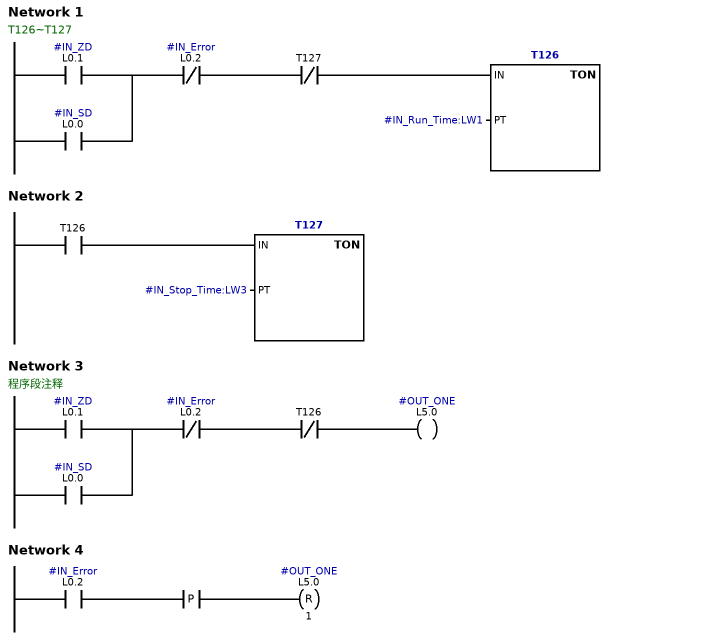
[picture p216: SBR112 networks 1-4]
Network 1
// T126~T127
LD     #IN_ZD:L0.1
O      #IN_SD:L0.0
AN     #IN_Error:L0.2
AN     T127
TON    T126, #IN_Run_Time:LW1
Network 2
LD     T126
TON    T127, #IN_Stop_Time:LW3
Network 3
// 程序段注释
LD     #IN_ZD:L0.1
O      #IN_SD:L0.0
AN     #IN_Error:L0.2
AN     T126
=      #OUT_ONE:L5.0
Network 4
LD     #IN_Error:L0.2
EU
R      #OUT_ONE:L5.0, 1
END_SUBROUTINE_BLOCK

SUBROUTINE_BLOCK Valve1_XH14:SBR113
TITLE=
VAR_INPUT
IN_SD:BOOL;	// L0.0 
IN_ZD:BOOL;	// L0.1 
IN_Error:BOOL;	// L0.2 
IN_Run_Time:INT;	// LW1 
IN_Stop_Time:INT;	// LW3 
END_VAR
VAR_OUTPUT
OUT_ONE:BOOL;	// L5.0 
END_VAR
VAR
TP1:BOOL;	// L5.1 
TP2:BOOL;	// L5.2 
END_VAR
BEGIN
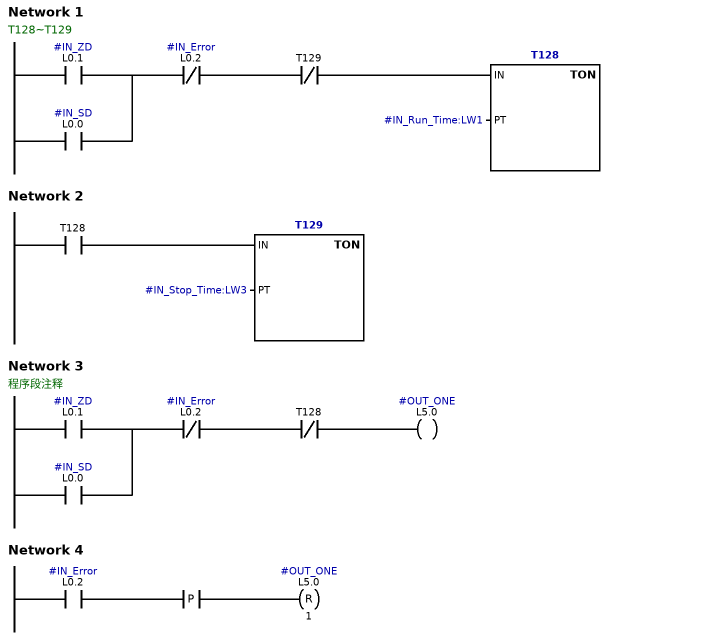
Network 1
// T128~T129
LD     #IN_ZD:L0.1
O      #IN_SD:L0.0
AN     #IN_Error:L0.2
AN     T129
TON    T128, #IN_Run_Time:LW1
Network 2
LD     T128
TON    T129, #IN_Stop_Time:LW3
Network 3
// 程序段注释
LD     #IN_ZD:L0.1
O      #IN_SD:L0.0
AN     #IN_Error:L0.2
AN     T128
=      #OUT_ONE:L5.0
Network 4
LD     #IN_Error:L0.2
EU
R      #OUT_ONE:L5.0, 1
END_SUBROUTINE_BLOCK

SUBROUTINE_BLOCK Valve1_XH15:SBR114
TITLE=
VAR_INPUT
IN_SD:BOOL;	// L0.0 
IN_ZD:BOOL;	// L0.1 
IN_Error:BOOL;	// L0.2 
IN_Run_Time:INT;	// LW1 
IN_Stop_Time:INT;	// LW3 
END_VAR
VAR_OUTPUT
OUT_ONE:BOOL;	// L5.0 
END_VAR
VAR
TP1:BOOL;	// L5.1 
TP2:BOOL;	// L5.2 
END_VAR
BEGIN
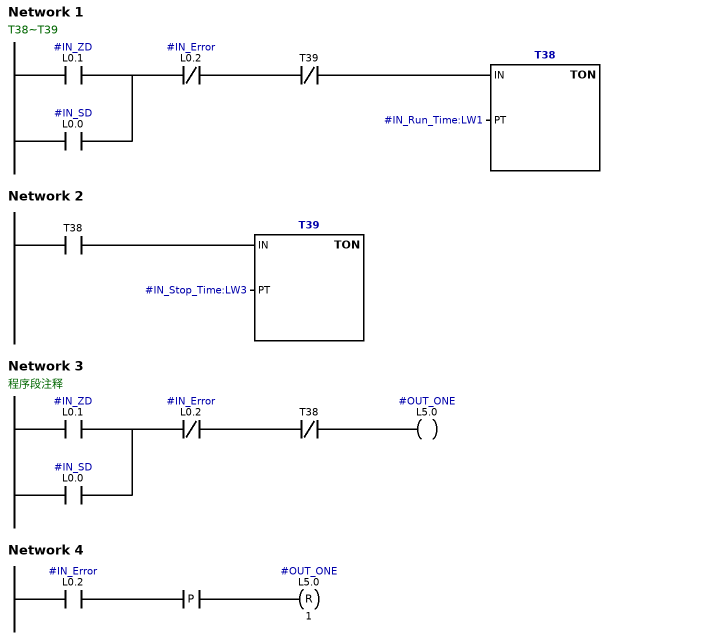
Network 1
// T38~T39  
LD     #IN_ZD:L0.1
O      #IN_SD:L0.0
AN     #IN_Error:L0.2
AN     T39
TON    T38, #IN_Run_Time:LW1
Network 2
LD     T38
TON    T39, #IN_Stop_Time:LW3
Network 3
// 程序段注释
LD     #IN_ZD:L0.1
O      #IN_SD:L0.0
AN     #IN_Error:L0.2
AN     T38
=      #OUT_ONE:L5.0
Network 4
LD     #IN_Error:L0.2
EU
R      #OUT_ONE:L5.0, 1
END_SUBROUTINE_BLOCK

SUBROUTINE_BLOCK Valve1_XH16:SBR115
TITLE=
VAR_INPUT
IN_SD:BOOL;	// L0.0 
IN_ZD:BOOL;	// L0.1 
IN_Error:BOOL;	// L0.2 
IN_Run_Time:INT;	// LW1 
IN_Stop_Time:INT;	// LW3 
END_VAR
VAR_OUTPUT
OUT_ONE:BOOL;	// L5.0 
END_VAR
VAR
TP1:BOOL;	// L5.1 
TP2:BOOL;	// L5.2 
END_VAR
BEGIN
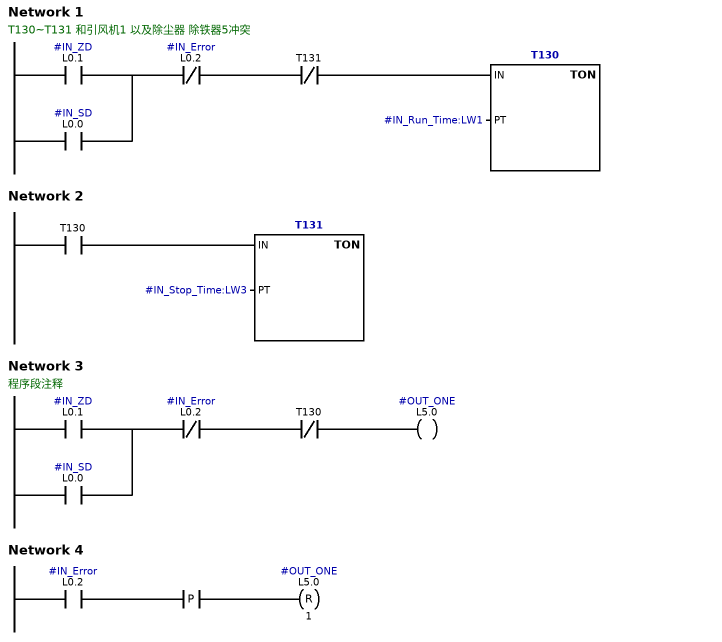
Network 1
// T130~T131 和引风机1 以及除尘器 除铁器5冲突
LD     #IN_ZD:L0.1
O      #IN_SD:L0.0
AN     #IN_Error:L0.2
AN     T131
TON    T130, #IN_Run_Time:LW1
Network 2
LD     T130
TON    T131, #IN_Stop_Time:LW3
Network 3
// 程序段注释
LD     #IN_ZD:L0.1
O      #IN_SD:L0.0
AN     #IN_Error:L0.2
AN     T130
=      #OUT_ONE:L5.0
Network 4
LD     #IN_Error:L0.2
EU
R      #OUT_ONE:L5.0, 1
END_SUBROUTINE_BLOCK

SUBROUTINE_BLOCK Valve1_XH17:SBR116
TITLE=
VAR_INPUT
IN_SD:BOOL;	// L0.0 
IN_ZD:BOOL;	// L0.1 
IN_Error:BOOL;	// L0.2 
IN_Run_Time:INT;	// LW1 
IN_Stop_Time:INT;	// LW3 
END_VAR
VAR_OUTPUT
OUT_ONE:BOOL;	// L5.0 
END_VAR
VAR
TP1:BOOL;	// L5.1 
TP2:BOOL;	// L5.2 
END_VAR
BEGIN
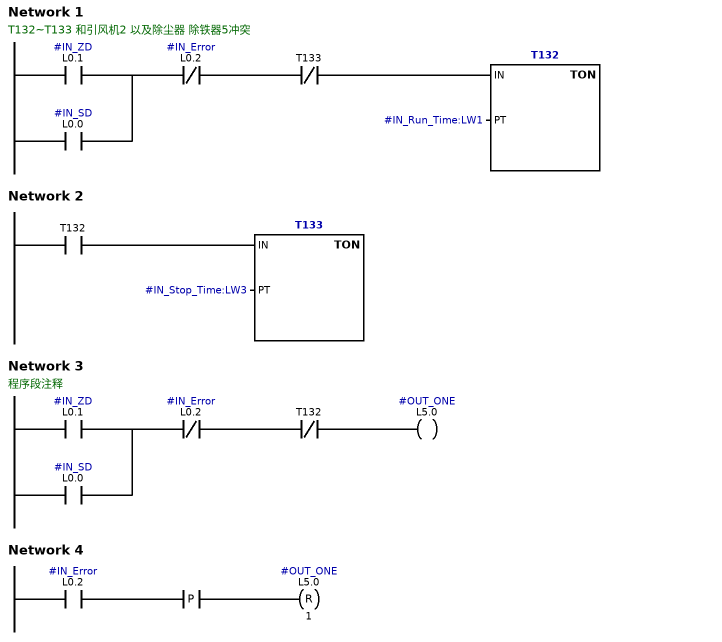
Network 1
// T132~T133 和引风机2 以及除尘器 除铁器5冲突
LD     #IN_ZD:L0.1
O      #IN_SD:L0.0
AN     #IN_Error:L0.2
AN     T133
TON    T132, #IN_Run_Time:LW1
Network 2
LD     T132
TON    T133, #IN_Stop_Time:LW3
Network 3
// 程序段注释
LD     #IN_ZD:L0.1
O      #IN_SD:L0.0
AN     #IN_Error:L0.2
AN     T132
=      #OUT_ONE:L5.0
Network 4
LD     #IN_Error:L0.2
EU
R      #OUT_ONE:L5.0, 1
END_SUBROUTINE_BLOCK

SUBROUTINE_BLOCK Valve1_XH18:SBR117
TITLE=
VAR_INPUT
IN_SD:BOOL;	// L0.0 
IN_ZD:BOOL;	// L0.1 
IN_Error:BOOL;	// L0.2 
IN_Run_Time:INT;	// LW1 
IN_Stop_Time:INT;	// LW3 
END_VAR
VAR_OUTPUT
OUT_ONE:BOOL;	// L5.0 
END_VAR
VAR
TP1:BOOL;	// L5.1 
TP2:BOOL;	// L5.2 
END_VAR
BEGIN
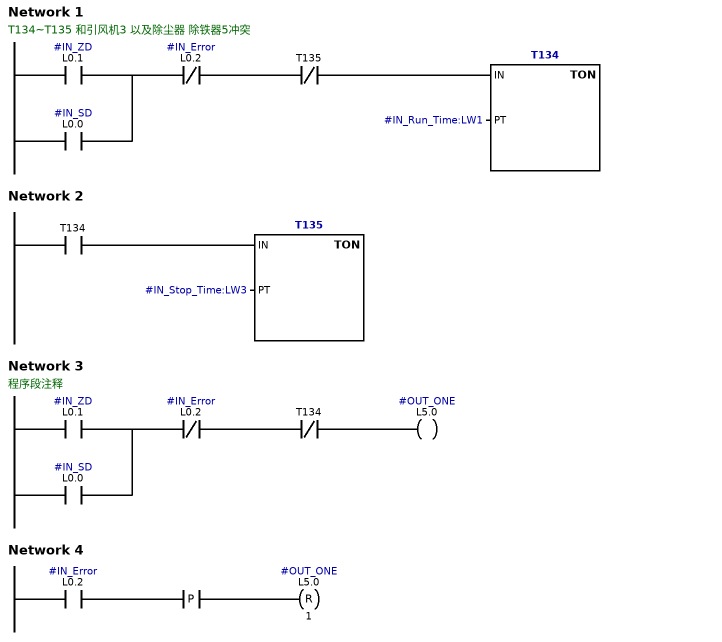
Network 1
// T134~T135 和引风机3 以及除尘器 除铁器5冲突
LD     #IN_ZD:L0.1
O      #IN_SD:L0.0
AN     #IN_Error:L0.2
AN     T135
TON    T134, #IN_Run_Time:LW1
Network 2
LD     T134
TON    T135, #IN_Stop_Time:LW3
Network 3
// 程序段注释
LD     #IN_ZD:L0.1
O      #IN_SD:L0.0
AN     #IN_Error:L0.2
AN     T134
=      #OUT_ONE:L5.0
Network 4
LD     #IN_Error:L0.2
EU
R      #OUT_ONE:L5.0, 1
END_SUBROUTINE_BLOCK

SUBROUTINE_BLOCK Valve1_XH19:SBR118
TITLE=
VAR_INPUT
IN_SD:BOOL;	// L0.0 
IN_ZD:BOOL;	// L0.1 
IN_Error:BOOL;	// L0.2 
IN_Run_Time:INT;	// LW1 
IN_Stop_Time:INT;	// LW3 
END_VAR
VAR_OUTPUT
OUT_ONE:BOOL;	// L5.0 
END_VAR
VAR
TP1:BOOL;	// L5.1 
TP2:BOOL;	// L5.2 
END_VAR
BEGIN
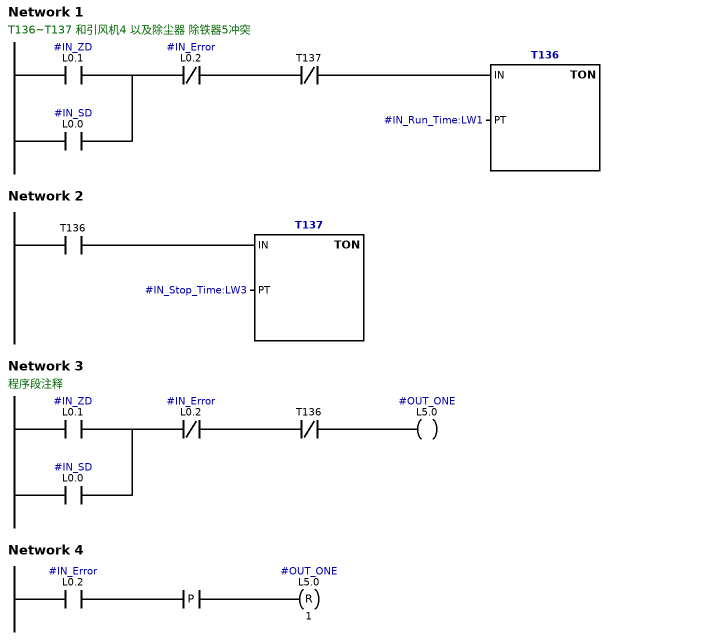
Network 1
// T136~T137 和引风机4 以及除尘器 除铁器5冲突
LD     #IN_ZD:L0.1
O      #IN_SD:L0.0
AN     #IN_Error:L0.2
AN     T137
TON    T136, #IN_Run_Time:LW1
Network 2
LD     T136
TON    T137, #IN_Stop_Time:LW3
Network 3
// 程序段注释
LD     #IN_ZD:L0.1
O      #IN_SD:L0.0
AN     #IN_Error:L0.2
AN     T136
=      #OUT_ONE:L5.0
Network 4
LD     #IN_Error:L0.2
EU
R      #OUT_ONE:L5.0, 1
END_SUBROUTINE_BLOCK

SUBROUTINE_BLOCK Valve1_XH20:SBR119
TITLE=
VAR_INPUT
IN_SD:BOOL;	// L0.0 
IN_ZD:BOOL;	// L0.1 
IN_Error:BOOL;	// L0.2 
IN_Run_Time:INT;	// LW1 
IN_Stop_Time:INT;	// LW3 
END_VAR
VAR_OUTPUT
OUT_ONE:BOOL;	// L5.0 
END_VAR
VAR
TP1:BOOL;	// L5.1 
TP2:BOOL;	// L5.2 
END_VAR
BEGIN
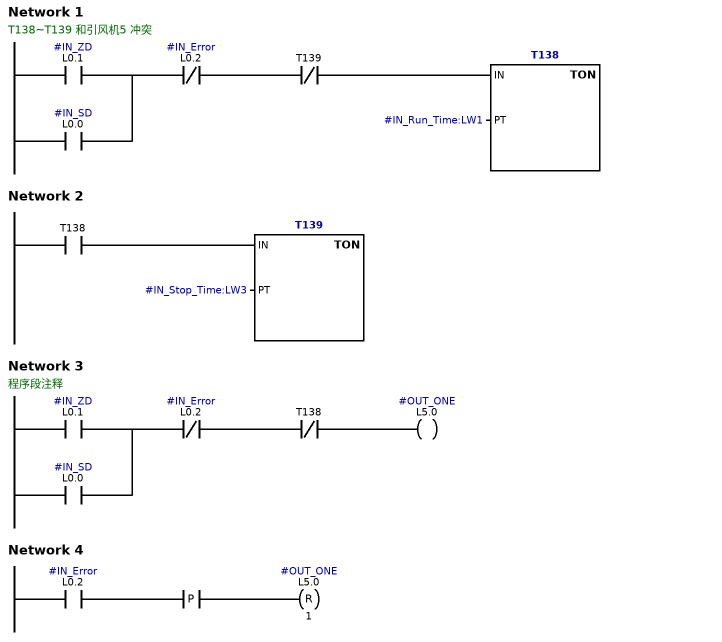
Network 1
// T138~T139 和引风机5 冲突
LD     #IN_ZD:L0.1
O      #IN_SD:L0.0
AN     #IN_Error:L0.2
AN     T139
TON    T138, #IN_Run_Time:LW1
Network 2
LD     T138
TON    T139, #IN_Stop_Time:LW3
Network 3
// 程序段注释
LD     #IN_ZD:L0.1
O      #IN_SD:L0.0
AN     #IN_Error:L0.2
AN     T138
=      #OUT_ONE:L5.0
Network 4
LD     #IN_Error:L0.2
EU
R      #OUT_ONE:L5.0, 1
END_SUBROUTINE_BLOCK

SUBROUTINE_BLOCK Valve2_XH1:SBR122
TITLE=
VAR_INPUT
IN_SD:BOOL;	// L0.0 
IN_ZD:BOOL;	// L0.1 
IN_Error:BOOL;	// L0.2 
IN_Run_Time:INT;	// LW1 
IN_Stop_Time:INT;	// LW3 
END_VAR
VAR_IN_OUT
TP1:BOOL;	// L5.0 
END_VAR
VAR_OUTPUT
OUT_1:BOOL;	// L5.1 
OUT_2:BOOL;	// L5.2 
END_VAR
VAR
TP2:BOOL;	// L5.3 
END_VAR
BEGIN
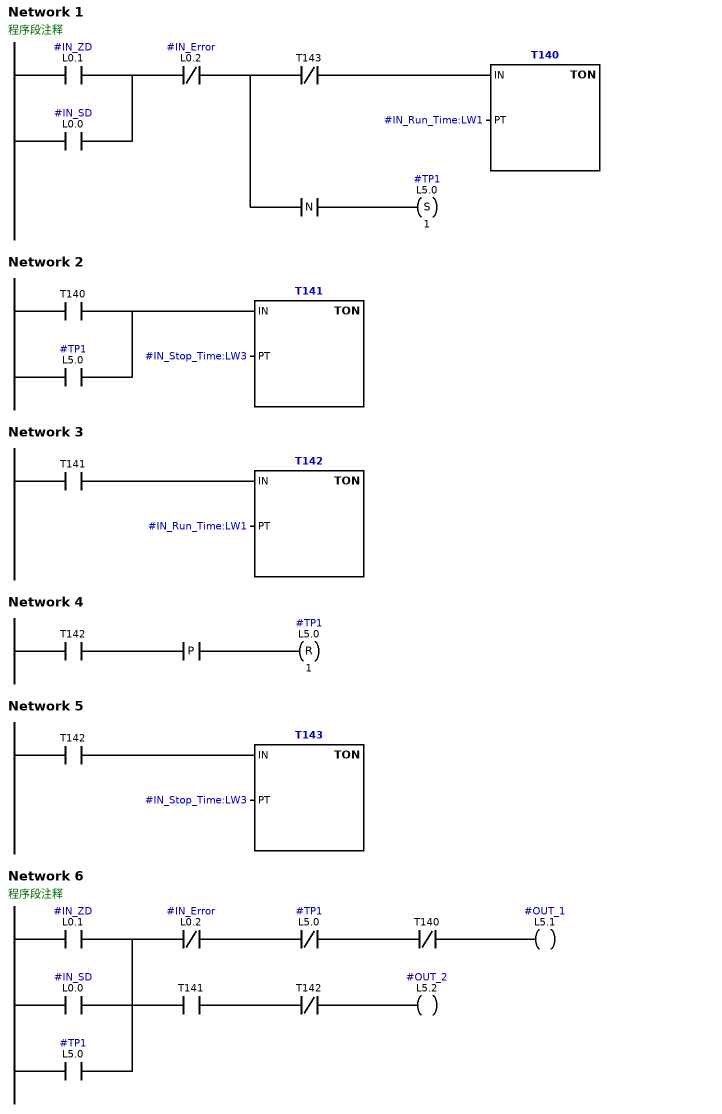
Network 1
// 程序段注释
LD     #IN_ZD:L0.1
O      #IN_SD:L0.0
AN     #IN_Error:L0.2
LPS
AN     T143
TON    T140, #IN_Run_Time:LW1
LPP
ED
S      #TP1:L5.0, 1
Network 2
LD     T140
O      #TP1:L5.0
TON    T141, #IN_Stop_Time:LW3
Network 3
LD     T141
TON    T142, #IN_Run_Time:LW1
Network 4
LD     T142
EU
R      #TP1:L5.0, 1
Network 5
LD     T142
TON    T143, #IN_Stop_Time:LW3
Network 6
// 程序段注释
LD     #IN_ZD:L0.1
O      #IN_SD:L0.0
O      #TP1:L5.0
LPS
AN     #IN_Error:L0.2
AN     #TP1:L5.0
AN     T140
=      #OUT_1:L5.1
LPP
A      T141
AN     T142
=      #OUT_2:L5.2
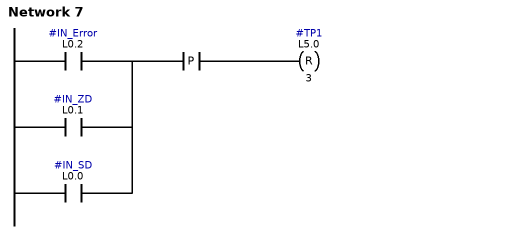
Network 7
LD     #IN_Error:L0.2
O      #IN_ZD:L0.1
O      #IN_SD:L0.0
EU
R      #TP1:L5.0, 3
END_SUBROUTINE_BLOCK

SUBROUTINE_BLOCK Valve2_XH2:SBR123
TITLE=
VAR_INPUT
IN_SD:BOOL;	// L0.0 
IN_ZD:BOOL;	// L0.1 
IN_Error:BOOL;	// L0.2 
IN_Run_Time:INT;	// LW1 
IN_Stop_Time:INT;	// LW3 
END_VAR
VAR_IN_OUT
TP1:BOOL;	// L5.0 
END_VAR
VAR_OUTPUT
OUT_1:BOOL;	// L5.1 
OUT_2:BOOL;	// L5.2 
END_VAR
VAR
TP2:BOOL;	// L5.3 
END_VAR
BEGIN
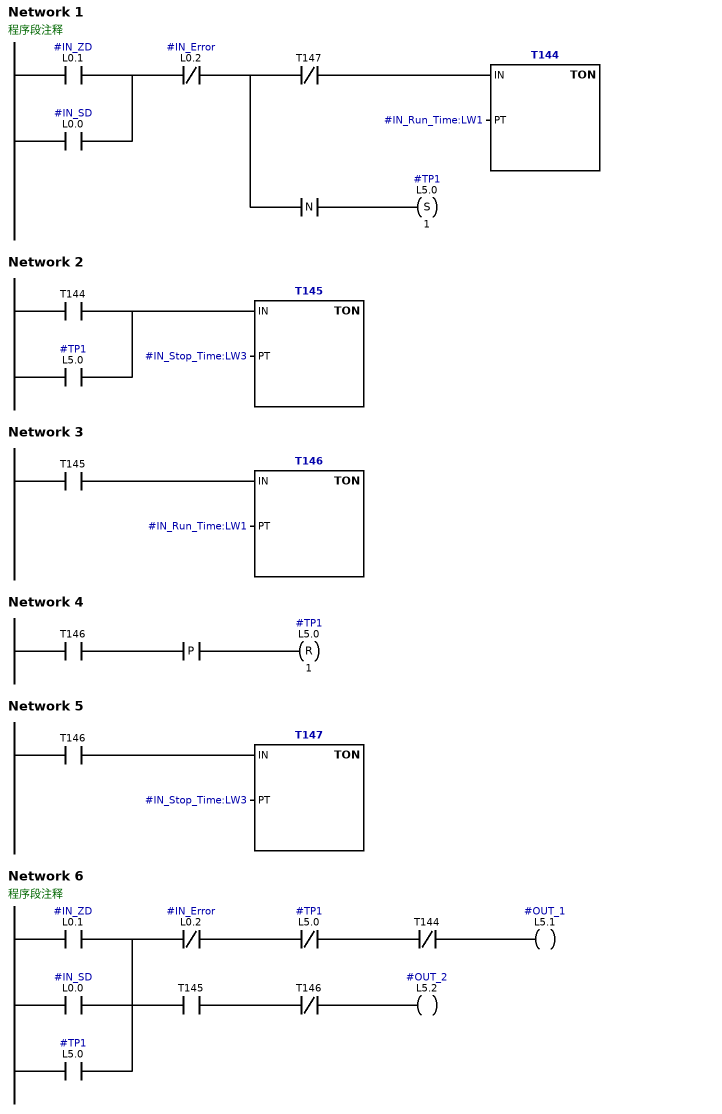
Network 1
// 程序段注释
LD     #IN_ZD:L0.1
O      #IN_SD:L0.0
AN     #IN_Error:L0.2
LPS
AN     T147
TON    T144, #IN_Run_Time:LW1
LPP
ED
S      #TP1:L5.0, 1
Network 2
LD     T144
O      #TP1:L5.0
TON    T145, #IN_Stop_Time:LW3
Network 3
LD     T145
TON    T146, #IN_Run_Time:LW1
Network 4
LD     T146
EU
R      #TP1:L5.0, 1
Network 5
LD     T146
TON    T147, #IN_Stop_Time:LW3
Network 6
// 程序段注释
LD     #IN_ZD:L0.1
O      #IN_SD:L0.0
O      #TP1:L5.0
LPS
AN     #IN_Error:L0.2
AN     #TP1:L5.0
AN     T144
=      #OUT_1:L5.1
LPP
A      T145
AN     T146
=      #OUT_2:L5.2
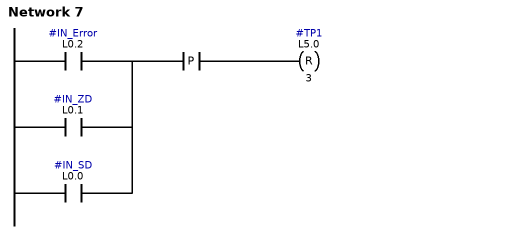
Network 7
LD     #IN_Error:L0.2
O      #IN_ZD:L0.1
O      #IN_SD:L0.0
EU
R      #TP1:L5.0, 3
END_SUBROUTINE_BLOCK

SUBROUTINE_BLOCK Valve2_XH3:SBR124
TITLE=
VAR_INPUT
IN_SD:BOOL;	// L0.0 
IN_ZD:BOOL;	// L0.1 
IN_Error:BOOL;	// L0.2 
IN_Run_Time:INT;	// LW1 
IN_Stop_Time:INT;	// LW3 
END_VAR
VAR_IN_OUT
TP1:BOOL;	// L5.0 
END_VAR
VAR_OUTPUT
OUT_1:BOOL;	// L5.1 
OUT_2:BOOL;	// L5.2 
END_VAR
VAR
TP2:BOOL;	// L5.3 
END_VAR
BEGIN
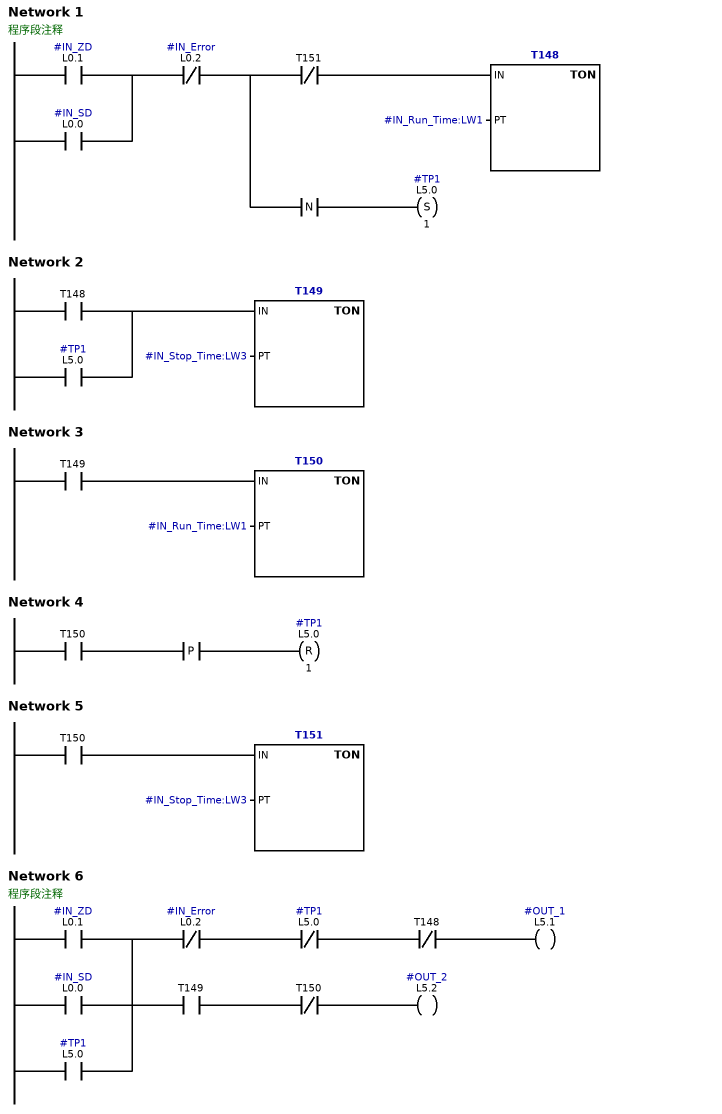
Network 1
// 程序段注释
LD     #IN_ZD:L0.1
O      #IN_SD:L0.0
AN     #IN_Error:L0.2
LPS
AN     T151
TON    T148, #IN_Run_Time:LW1
LPP
ED
S      #TP1:L5.0, 1
Network 2
LD     T148
O      #TP1:L5.0
TON    T149, #IN_Stop_Time:LW3
Network 3
LD     T149
TON    T150, #IN_Run_Time:LW1
Network 4
LD     T150
EU
R      #TP1:L5.0, 1
Network 5
LD     T150
TON    T151, #IN_Stop_Time:LW3
Network 6
// 程序段注释
LD     #IN_ZD:L0.1
O      #IN_SD:L0.0
O      #TP1:L5.0
LPS
AN     #IN_Error:L0.2
AN     #TP1:L5.0
AN     T148
=      #OUT_1:L5.1
LPP
A      T149
AN     T150
=      #OUT_2:L5.2
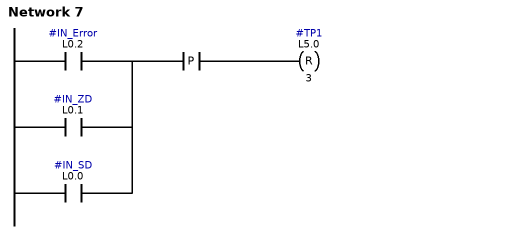
Network 7
LD     #IN_Error:L0.2
O      #IN_ZD:L0.1
O      #IN_SD:L0.0
EU
R      #TP1:L5.0, 3
END_SUBROUTINE_BLOCK

SUBROUTINE_BLOCK Valve2_XH4:SBR125
TITLE=
VAR_INPUT
IN_SD:BOOL;	// L0.0 
IN_ZD:BOOL;	// L0.1 
IN_Error:BOOL;	// L0.2 
IN_Run_Time:INT;	// LW1 
IN_Stop_Time:INT;	// LW3 
END_VAR
VAR_IN_OUT
TP1:BOOL;	// L5.0 
END_VAR
VAR_OUTPUT
OUT_1:BOOL;	// L5.1 
OUT_2:BOOL;	// L5.2 
END_VAR
VAR
TP2:BOOL;	// L5.3 
END_VAR
BEGIN
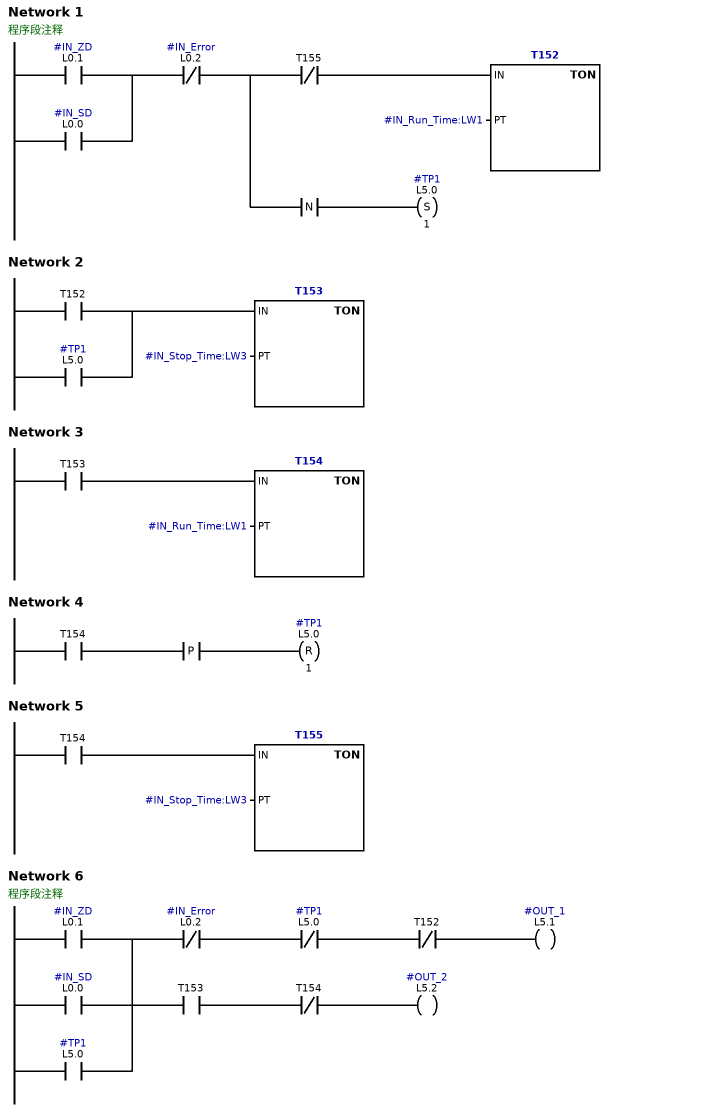
Network 1
// 程序段注释
LD     #IN_ZD:L0.1
O      #IN_SD:L0.0
AN     #IN_Error:L0.2
LPS
AN     T155
TON    T152, #IN_Run_Time:LW1
LPP
ED
S      #TP1:L5.0, 1
Network 2
LD     T152
O      #TP1:L5.0
TON    T153, #IN_Stop_Time:LW3
Network 3
LD     T153
TON    T154, #IN_Run_Time:LW1
Network 4
LD     T154
EU
R      #TP1:L5.0, 1
Network 5
LD     T154
TON    T155, #IN_Stop_Time:LW3
Network 6
// 程序段注释
LD     #IN_ZD:L0.1
O      #IN_SD:L0.0
O      #TP1:L5.0
LPS
AN     #IN_Error:L0.2
AN     #TP1:L5.0
AN     T152
=      #OUT_1:L5.1
LPP
A      T153
AN     T154
=      #OUT_2:L5.2
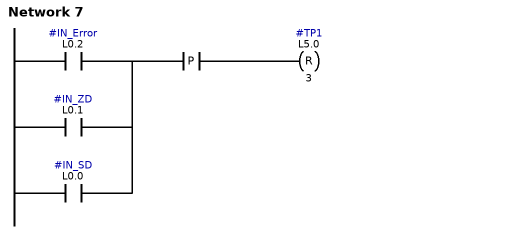
Network 7
LD     #IN_Error:L0.2
O      #IN_ZD:L0.1
O      #IN_SD:L0.0
EU
R      #TP1:L5.0, 3
END_SUBROUTINE_BLOCK

SUBROUTINE_BLOCK Valve2_XH5:SBR126
TITLE=
VAR_INPUT
IN_SD:BOOL;	// L0.0 
IN_ZD:BOOL;	// L0.1 
IN_Error:BOOL;	// L0.2 
IN_Run_Time:INT;	// LW1 
IN_Stop_Time:INT;	// LW3 
END_VAR
VAR_IN_OUT
TP1:BOOL;	// L5.0 
END_VAR
VAR_OUTPUT
OUT_1:BOOL;	// L5.1 
OUT_2:BOOL;	// L5.2 
END_VAR
VAR
TP2:BOOL;	// L5.3 
END_VAR
BEGIN
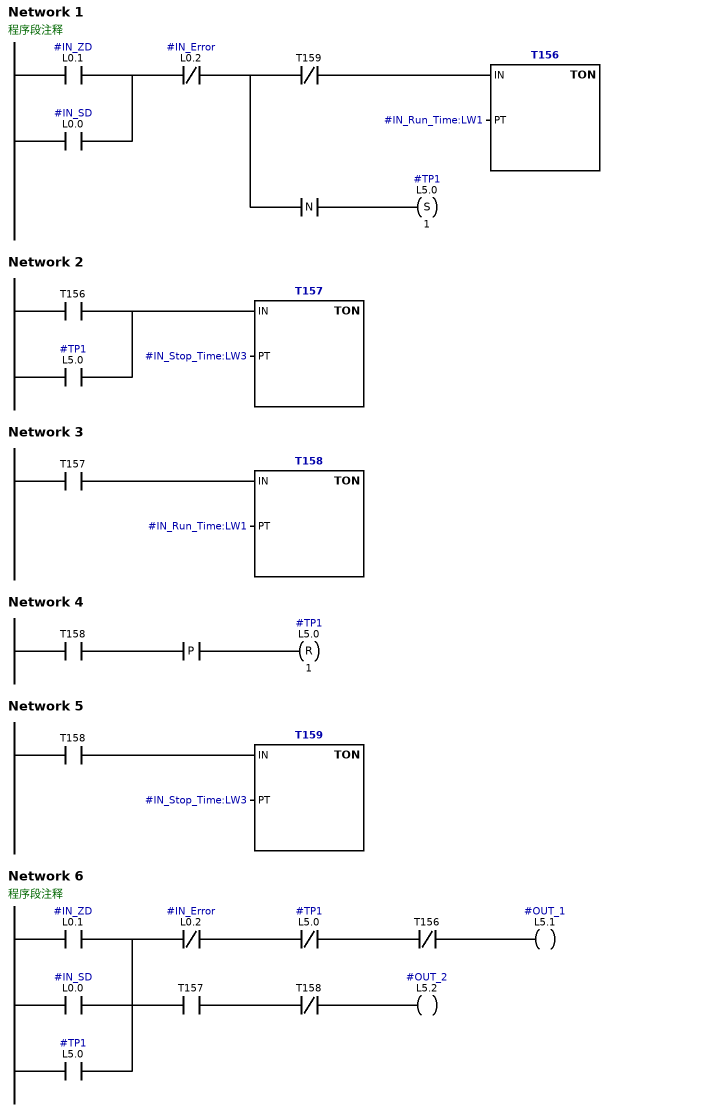
Network 1
// 程序段注释
LD     #IN_ZD:L0.1
O      #IN_SD:L0.0
AN     #IN_Error:L0.2
LPS
AN     T159
TON    T156, #IN_Run_Time:LW1
LPP
ED
S      #TP1:L5.0, 1
Network 2
LD     T156
O      #TP1:L5.0
TON    T157, #IN_Stop_Time:LW3
Network 3
LD     T157
TON    T158, #IN_Run_Time:LW1
Network 4
LD     T158
EU
R      #TP1:L5.0, 1
Network 5
LD     T158
TON    T159, #IN_Stop_Time:LW3
Network 6
// 程序段注释
LD     #IN_ZD:L0.1
O      #IN_SD:L0.0
O      #TP1:L5.0
LPS
AN     #IN_Error:L0.2
AN     #TP1:L5.0
AN     T156
=      #OUT_1:L5.1
LPP
A      T157
AN     T158
=      #OUT_2:L5.2
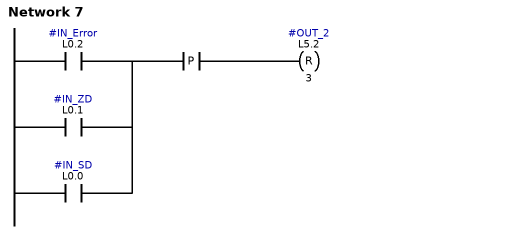
Network 7
LD     #IN_Error:L0.2
O      #IN_ZD:L0.1
O      #IN_SD:L0.0
EU
R      #OUT_2:L5.2, 3
END_SUBROUTINE_BLOCK

DATA_BLOCK_TAB 页面_1
BEGIN
         Time1, 50
         Time2, 50
         Time3, 50
         Time4, 50
         Time5, 50
         Time6, 50
         Time7, 50
         Time8, 50
         Time9, 50
         Time10, 50
         Time11, 50
         Time12, 50
         Time13, 50
         Time14, 50
         Time15, 50
         Time16, 50
         Time17, 50
         Time18, 50
         Time19, 50
         Time20, 50
         Time21, 50
         Time22, 50
         Time23, 50
         Time24, 50
         Time25, 50
         Time26, 50
         Time27, 50
         Time28, 50
         Time29, 50
         Time30, 50
         Time31, 50
         Time32, 50
         Time33, 50
         Time34, 50
         Time35, 50
         Time36, 50
         Time37, 50
         Time38, 50
         Time39, 50
         Time40, 50
         Time41, 50
         Time42, 50
         Time43, 50
         Time44, 50
         Time45, 50
         Time46, 50
         Time47, 50
         Time48, 50
         Time49, 50
         Time50, 50
         Time51, 50
         Time52, 50
         Time53, 50
         Time54, 50
         Time55, 50
         Time56, 50
         Time57, 50
         Time58, 50
         Time59, 50
         Time60, 50
         Time61, 50
         Time62, 50
         Time63, 50
         Time64, 50
         Time65, 50
         Time66, 50
         Time67, 50
         Time68, 50
         Time69, 50
         Time70, 50
         Time71, 50
         Time72, 50
         Time73, 50
         Time74, 50
         Time75, 50
         Time76, 50
         Time77, 50
         Time78, 50
         Time79, 50
         Time80, 50
         Time81, 50
         Time82, 50
         Time83, 50
         Time84, 50
         Time85, 50
         Time86, 50
         Time87, 50
         Time88, 50
         Time89, 50
         Time90, 50
         Time91, 50
         Time92, 50
         Time93, 50
         Time94, 50
         Time95, 50
         Time96, 50
         Time97, 50
         Time98, 50
         Time99, 50
         Time100, 50
         Time101, 50
         Time102, 50
         Time103, 50
         Time104, 50
         Time105, 50
         Time106, 50
         Time107, 50
         Time108, 50
         Time109, 50
         Time110, 50
         Time111, 50
         Time112, 50
         Time113, 50
         Time114, 50
         Time115, 50
         Time116, 50
         Time117, 50
         Time118, 50
         Time119, 50
         Time120, 50
         Time121, 50
         Time122, 50
         Time123, 50
         Time124, 50
         Time125, 50
         Time126, 50
         Time127, 50
         Time128, 50
         Time129, 50
         Time130, 50
         Time131, 50
         Time132, 50
         Time133, 50
         Time134, 50
         Time135, 50
         Time136, 50
         Time137, 50
         Time138, 50
         Time139, 50
         Time140, 50
         Time141, 50
         Time142, 50
         Time143, 50
         Time144, 50
         Time145, 50
         Time146, 50
         Time147, 50
         Time148, 50
         Time149, 50
         Time150, 50
         AI_Sst_H0, 3000.0
         AI_Sst_H1, 3000.0
         AI_Sst_H2, 3000.0
         AI_Sst_H3, 3000.0
         AI_Sst_H4, 3000.0
         AI_Sst_H5, 3000.0
         AI_Sst_H6, 3000.0
         AI_Sst_H7, 3000.0
         AI_Sst_H8, 3000.0
         AI_Sst_H9, 3000.0
         AI_Sst_H10, 3000.0
         AI_Sst_H11, 3000.0
         AI_Sst_H12, 3000.0
         AI_Sst_H13, 3000.0
         AI_Sst_H14, 3000.0
         AI_Sst_H15, 3000.0
         AI_Sst_H16, 3000.0
         AI_Sst_H17, 3000.0
         AI_Sst_H18, 3000.0
         AI_Sst_H19, 3000.0
         AI_Sst_H20, 3000.0
         AI_Sst_H21, 3000.0
         AI_Sst_H22, 3000.0
         AI_Sst_H23, 3000.0
         AI_Sst_H24, 3000.0
         AI_BJ_0, 1500.0
         AI_BJ_1, 1500.0
         AI_BJ_2, 1500.0
         AI_BJ_3, 1500.0
         AI_BJ_4, 1500.0
         AI_BJ_5, 1500.0
         AI_BJ_6, 1500.0
         AI_BJ_7, 1500.0
         AI_BJ_8, 1500.0
         AI_BJ_9, 1500.0
         AI_BJ_10, 1500.0
         AI_BJ_11, 1500.0
         AI_BJ_12, 1500.0
         AI_BJ_13, 1500.0
         AI_BJ_14, 1500.0
         AI_BJ_15, 1500.0
         AI_BJ_16, 1500.0
         AI_BJ_17, 1500.0
         AI_BJ_18, 1500.0
         AI_BJ_19, 1500.0
         AI_BJ_20, 1500.0
         AI_BJ_21, 1500.0
         AI_BJ_22, 1500.0
         AI_BJ_23, 1500.0
         AI_BJ_24, 1500.0
         AI_TJ_0, 2000.0
         AI_TJ_1, 2000.0
         AI_TJ_2, 2000.0
         AI_TJ_3, 2000.0
         AI_TJ_4, 2000.0
         AI_TJ_5, 2000.0
         AI_TJ_6, 2000.0
         AI_TJ_7, 2000.0
         AI_TJ_8, 2000.0
         AI_TJ_9, 2000.0
         AI_TJ_10, 2000.0
         AI_TJ_11, 2000.0
         AI_TJ_12, 2000.0
         AI_TJ_13, 2000.0
         AI_TJ_14, 2000.0
         AI_TJ_15, 2000.0
         AI_TJ_16, 2000.0
         AI_TJ_17, 2000.0
         AI_TJ_18, 2000.0
         AI_TJ_19, 2000.0
         AI_TJ_20, 2000.0
         AI_TJ_21, 2000.0
         AI_TJ_22, 2000.0
         AI_TJ_23, 2000.0
         AI_TJ_24, 2000.0
         Set_INT_0, 20
         Set_INT_1, 20
         Set_INT_2, 20
         Set_INT_3, 20
         Set_INT_4, 20
         Set_INT_5, 20
         Set_INT_6, 20
         Set_INT_7, 20
         Set_INT_8, 20
         Set_INT_9, 20
         Set_INT_10, 20
         Set_INT_11, 20
         Set_INT_12, 20
         Set_INT_13, 20
         Set_INT_14, 20
         Set_R0, 30.0
         Set_R1, 30.0
         Set_R2, 30.0
         Set_R3, 30.0
         Set_R4, 30.0
         Set_R5, 30.0
         Set_R6, 30.0
         Set_R7, 30.0
         Set_R8, 30.0
         Set_R9, 30.0
         Set_R10, 30.0
         Set_R11, 30.0
         Set_R12, 30.0
         Set_R13, 30.0
         Set_R14, 30.0
         Set_R15, 30.0
         Set_R16, 30.0
         Set_R17, 30.0
         Set_R18, 30.0
         Set_R19, 30.0
         Set_R20, 30.0
         Set_R21, 30.0
         Set_R22, 30.0
         Set_R23, 30.0
         Set_R24, 30.0
         仓泵1压力低于, 30.0
         仓泵2压力低于, 30.0
         仓泵3压力低于, 30.0
         仓泵4压力低于, 30.0
         仓泵5压力低于, 30.0
         除尘器1切换值, 300.0
         除尘器2切换值, 300.0
         除尘器3切换值, 300.0
         除尘器4切换值, 300.0
         除尘器5切换值, 300.0
         称重1切换值, 300.0
         称重2切换值, 300.0
         称重3切换值, 300.0
         称重4切换值, 300.0
         称重5切换值, 300.0
         除尘器1设定时间, 36
         除尘器2设定时间, 42
         除尘器3设定时间, 48
         除尘器4设定时间, 54
         除尘器5设定时间, 60
         反打1设定时间, 36
         反打2设定时间, 42
         反打3设定时间, 48
         反打4设定时间, 54
         反打5设定时间, 60
END_DATA_BLOCK_TAB
